// TIA Portal V20 export
FUNCTION "CallSimulation" : Void   // FC22, LAD
TITLE = CallSimulation
// This blocks switches between simulation with SIMIT and PLCSIM Advanced or with PLCSIM and PLC internal simulation function blocks
// stored: IsIECCheckEnabled true, SetENOAutomatically true
BEGIN
END_FUNCTION
